SUBAPPLICATION INI_OPC_PARAM (* OPC_UA Parameter lesen Schreiben. *)
  (* Standard: 61499-2; Description: Copyright (c) 2023 Meisterschulen am Ostbahnhof This program and the accompanying materials are made available under the terms of the Eclipse Public License 2.0 which is available at https://www.eclipse.org/legal/epl-2.0/ SPDX-License-Identifier: EPL-2.0 *)
  (* Version 1.1, 2026-07-20, Franz Höpfinger, Meisterschulen am Ostbahnhof, Background *)
  (* Version 1.0, 2026-01-15, Franz Höpfinger, Meisterschulen am Ostbahnhof, initial API and implementation and/or initial documentation *)
  PACKAGE MyLib::sys;
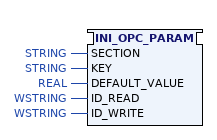
  VAR_INPUT
    SECTION : STRING; (* INI-Abschnitt (settings.ini) *)
    KEY : STRING; (* INI-Schluessel innerhalb SECTION *)
    DEFAULT_VALUE : REAL; (* Wert falls in settings.ini nicht vorhanden *)
    ID_READ : WSTRING; (* OPC-UA-Verbindungsstring (READ) - Client schreibt hier einen neuen Wert *)
    ID_WRITE : WSTRING; (* OPC-UA-Verbindungsstring (WRITE) - aktuell gespeicherter Wert wird hier publiziert *)
  END_VAR
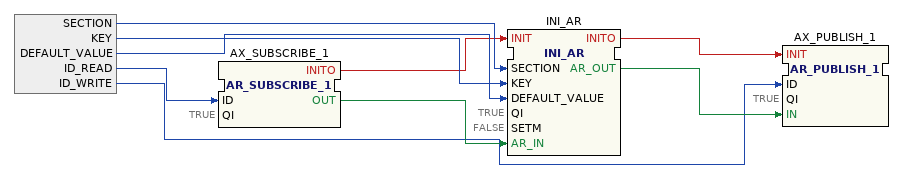
  FBS
    AX_SUBSCRIBE_1 : adapter::net::AR_SUBSCRIBE_1(QI := TRUE);
    AX_PUBLISH_1 : adapter::net::AR_PUBLISH_1(QI := TRUE);
    INI_AR : eclipse4diac::storage::INI_AR(QI := TRUE, SETM := FALSE);
  END_FBS
  EVENT_CONNECTIONS
    AX_SUBSCRIBE_1.INITO TO INI_AR.INIT;
    INI_AR.INITO TO AX_PUBLISH_1.INIT;
  END_CONNECTIONS
  DATA_CONNECTIONS
    SECTION TO INI_AR.SECTION;
    KEY TO INI_AR.KEY;
    DEFAULT_VALUE TO INI_AR.DEFAULT_VALUE;
    ID_READ TO AX_SUBSCRIBE_1.ID;
    ID_WRITE TO AX_PUBLISH_1.ID;
  END_CONNECTIONS
  ADAPTER_CONNECTIONS
    AX_SUBSCRIBE_1.OUT TO INI_AR.AR_IN;
    INI_AR.AR_OUT TO AX_PUBLISH_1.IN;
  END_CONNECTIONS
END_SUBAPPLICATION
